(* IEC 61131-3 sources: MsgBoxErr/, 2 files *)

(* ---- MsgBoxAck.st ---- *)
(********************************************************************
 * COPYRIGHT --
 ********************************************************************
 * Program: RecipeUpdater
 * File: MsgBoxAck.st
 * Author: Josh
 * Created: July 14, 2015
 ********************************************************************
 * Implementation of program RecipeUpdater
 ********************************************************************)

(* This function block will post a message block that can be acknowledged or add to the error collector *)
FUNCTION_BLOCK MsgBoxAck

	IF AckError THEN
		AckError:= FALSE;
		Accept:=	FALSE;
		Ignored:=	FALSE;
		ErrorTimeout.IN:=	TRUE;
	END_IF

	//Give an acknowledge error some time to clear
	ErrorTimeout.PT:=	T#1s;
	ErrorTimeout();
	IF ErrorTimeout.Q THEN
		ErrorTimeout.IN:=	FALSE;
		ErrorAdded:= FALSE;
	END_IF

	Execute:= 	FALSE;

	IF Active
		AND MsgID = 0
		AND NOT Ignored
		THEN

		OkAddr:=0;
		IgnoreAddr:=0;

		IF OKText <> '' THEN
			OkAddr:=ADR(OKText);
			OkCmd:=ADR(Accept);
		END_IF
		IF IgnoreText <> '' THEN
			IgnoreAddr:=ADR(IgnoreText);
			IgnoreCmd:=	ADR(Ignored);
		END_IF

		IF Password = '' THEN
			MsgID:= MessageBox_AddMsg(ADR(Message),OkAddr,OkCmd,IgnoreAddr,IgnoreCmd);
		ELSE
			InputPassword:='';
			MsgID:= PromptBox_AddMsg(ADR(Message),ADR(InputPassword),OkAddr,OkCmd,IgnoreAddr,IgnoreCmd);
		END_IF
	ELSIF NOT Active THEN
		Ignored:=0;
		Accept:=0;
	END_IF

	IF MsgID <> 0
		AND (NOT Active OR Ignored)
		THEN
		MessageBox_RemoveMsg(MsgID);
		MsgID:=	0;
	END_IF

	IF (Password <> '' AND Ignored) OR (IsError AND Active)
		THEN
		IF NOT ErrorAdded THEN
			IF pErrCol <> 0 THEN
				dErrcol ACCESS pErrCol;
				addstatus:=errcolAddError(ADR(''),ADR(Message),1,ADR(AckError),dErrcol);
				IF addstatus = 0 OR addstatus = 58202 THEN
					ErrorAdded:= TRUE;
				END_IF
			END_IF
		END_IF
	END_IF

	IF Accept THEN
		MsgID:=		0;
		Accept:=	0;
		Ignored:=	0;
		IF Password <> '' THEN
			IF Password = InputPassword THEN
				Execute:= 	TRUE;
			ELSE
				Ignored:= TRUE;
			END_IF
		ELSE
			Execute:= 	TRUE;
		END_IF
	END_IF

END_FUNCTION_BLOCK

(* ---- MsgBoxErr.fun ---- *)
FUNCTION_BLOCK MsgBoxAck (*TODO: Add your comment here*)
	VAR_INPUT
		Active : BOOL;
		IsError : BOOL;
		Message : STRING[320];
		OKText : STRING[20];
		IgnoreText : STRING[20];
		Password : STRING[80];
		pErrCol : UDINT;
	END_VAR
	VAR_OUTPUT
		Execute : BOOL;
		Ignored : BOOL;
	END_VAR
	VAR
		MsgID : UDINT;
		Accept : BOOL;
		AckError : BOOL;
		ErrorAdded : BOOL;
		InputPassword : STRING[80];
		dErrcol : REFERENCE TO ErrorCollector_typ;
		ErrorTimeout : TON;
		OkAddr : UDINT;
		OkCmd : UDINT;
		IgnoreAddr : UDINT;
		IgnoreCmd : UDINT;
		addstatus : UINT;
	END_VAR
END_FUNCTION_BLOCK
